PROGRAM FeedMotor1Manualcontrol
VAR
END_VAR
// Written 10.08.2023 by Daniel Kelly

// Program provides manual control of the motor M1 via its switch

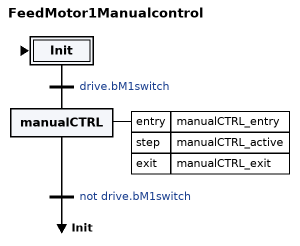
INITIAL_STEP Init:
END_STEP
TRANSITION FROM Init TO manualCTRL
    := drive.bM1switch;
END_TRANSITION
STEP manualCTRL:
    manualCTRL_entry(P1);  // entry action
    manualCTRL_active(N);  // step action
    manualCTRL_exit(P0);  // exit action
END_STEP
TRANSITION FROM manualCTRL TO Init
    := not drive.bM1switch;
END_TRANSITION

ACTION manualCTRL_active:
IF drive.ATV_TPDO_Input1_Status_Word = atv_status.rdy2SwitchON THEN 
	drive.ATV_RPDO_Output1_Control_Word := 7;
END_IF

IF drive.ATV_TPDO_Input1_Status_Word = atv_status.SwitchedON THEN 
	drive.ATV_RPDO_Output1_Control_Word := 15;
	drive.bM1active := TRUE; 
END_IF

drive.bFeedMotor2 := TRUE;
END_ACTION

ACTION manualCTRL_entry:
drive.ATV_RPDO_Output2_Target_Velocity := 1000;
drive.ATV_RPDO_Output1_Control_Word := 6;
END_ACTION

ACTION manualCTRL_exit:
drive.ATV_RPDO_Output1_Control_Word := 7; 
drive.bM1active := FALSE;

drive.bFeedMotor2 := FALSE;
END_ACTION

END_PROGRAM

(* stored: Version 1.1.0.1, ProductVersion 3.1.4024.12
   POU FeedMotor1Manualcontrol: Id {0363e149-5b31-4191-8a15-a5454c60392f}, SpecialFunc None
   Action manualCTRL_active: Id {2bce3834-f89a-4fbd-a0dc-57666f09bf32}
   Action manualCTRL_entry: Id {aef74774-bc2d-43e0-ab2e-4a459e0905f7}
   Action manualCTRL_exit: Id {834dae2d-8550-480f-96bd-3e97dea03069} *)
